Fanuc TP program (LS listing): Drop.LS

/PROG  DROP
/ATTR
OWNER		= MNEDITOR;
COMMENT		= "";
PROG_SIZE	= 306;
CREATE		= DATE 25-06-04  TIME 04:06:58;
MODIFIED	= DATE 25-06-04  TIME 04:06:58;
FILE_NAME	= ;
VERSION		= 0;
LINE_COUNT	= 5;
MEMORY_SIZE	= 658;
PROTECT		= READ_WRITE;
TCD:  STACK_SIZE	= 0,
      TASK_PRIORITY	= 50,
      TIME_SLICE	= 0,
      BUSY_LAMP_OFF	= 0,
      ABORT_REQUEST	= 0,
      PAUSE_REQUEST	= 0;
DEFAULT_GROUP	= 1,*,*,*,*;
CONTROL_CODE	= 00000000 00000000;
LOCAL_REGISTERS	= 0,0,0;
/MN
   1:  !FANUC America Corp. ;
   2:  !ROBOGUIDE Generated This TPP ;
   3:  !Run SimPRO.cf to setup frame and ;
   4:  ! Drop ('Part1') From ('GP: 1 - U ;
   5:  !WAIT 0.00 (sec) ;
/POS
/END
